FUNCTION_BLOCK FB_PrintPositionDmax EXTENDS FB_BasePrint IMPLEMENTS I_Sim
VAR_INPUT
  IlEncoderPulse      AT%I* : UDINT;                // Encoder counter intput
  IbEncoderWcState    AT%I* : BOOL;                 // Encoder EL5101 WcState
END_VAR
VAR_OUTPUT
  bStarted                  : BOOL;                 // position started moving
  bMoving                   : BOOL;                 // position is moving
END_VAR
// ----------------------------------
// configuration
VAR
  // configuration (init)
  _fPrintResolution         : LREAL := 600;         // print(head) resolution in [dpi]
  _fSubPxResolution         : LREAL := 32;          // SubPixel resolution [SubPx], resolution factor (fI_PrintResolution*fI_SubPxResolution=>Output resolution)
  _fTaskCycleTime           : LREAL := 0.002;        // Task cycle time in [s]
END_VAR
VAR PERSISTENT
  // config values changable during runtime (recipe, visu, property)
  _fEncoderResolution       : LREAL := 2.00475;     // Encoder resolution
  _bEnSpeedComp             : BOOL := FALSE;
  _fSpeedCompFactor         : LREAL := 0.0;         // TODO: define value
  _fSpeedCompRefSpeed       : LREAL := 0.0;         // TODO: define value
END_VAR
VAR CONSTANT
  fC_MinSpeed               : LREAL := 0.05;
END_VAR
// ---------------------------------
// internal variables
VAR
  // fb inst
  fbPositionMaster          : FB_PositionMaster;

  // internal vars
  fEncoderReso              : LREAL;                // used encoder resolution
  rTrigMoving               : R_TRIG;
  // simulation
  _bSim                     : BOOL;
    
  // test functions
  (*bEnTestVsOld              : BOOL;    
  fbVencoder                : FB_V_ENCODER;
  Fb_Ph_Master              : FB_POSITION_MASTER;
  *)
END_VAR

// set internal used resolution
fEncoderReso := _fEncoderResolution;  

// compensate resolution (if enabled)
IF _bEnSpeedComp THEN
  fEncoderReso := F_EncoderSpeedComp(   
    fMasterSpeed:=fbPositionMaster.fMasterSpeed,
    fResolution:=fEncoderReso,
    fSpeedCompFactor:=_fSpeedCompFactor,
    fSpeedCompRefSpeed:=_fSpeedCompRefSpeed
  );
END_IF

// calc position / speed
fbPositionMaster(fResolutionInput:=fEncoderReso, lPosReference:=IlEncoderPulse);
// postion status
bMoving := ABS(fbPositionMaster.fMasterSpeed) >= fC_MinSpeed; 
rTrigMoving(CLK:=bMoving);   // create started trigger output
bStarted := rTrigMoving.Q OR fbPositionMaster.bSyncReq;

{attribute 'monitoring' := 'call'}
(*Simulation is enabled set/get*)
PROPERTY bSimEnable : BOOL
GET
bSimEnable := _bSim;
END_GET
SET
_bSim := bSimEnable;
fbPositionMaster.bSim := _bSim;
END_SET
END_PROPERTY

(*
  Get current "default" position.
  [SubPx] as return value and [um] as output
  :return: position in SubPx resolution
*)
METHOD getPosition : DINT
VAR_OUTPUT
  nPosition_px       : DINT;                 // Master position in [px]
  fPosition_um       : LREAL;                // Master position in [um]
END_VAR
getPosition := fbPositionMaster.lMasterPosition;
nPosition_px := fbPositionMaster.lMasterPosition / LREAL_TO_DINT(_fSubPxResolution);
fPosition_um := fbPositionMaster.fMasterPosition;
END_METHOD

(*
  Get "default" speed.
*)
METHOD getSpeed : LREAL
getSpeed := fbPositionMaster.fMasterSpeed;
END_METHOD

METHOD Init : BOOL
VAR_INPUT
  fPrintResolution    : LREAL := 600;         // print(head) resolution in [dpi]
  fSubPxResolution    : LREAL := 32;          // SubPixel resolution [SubPx], resolution factor (fI_PrintResolution*fI_SubPxResolution=>Output resolution)
  fTaskCycleTime      : LREAL;                 // Task cycle time in [s]
END_VAR
// store config
_fPrintResolution := fPrintResolution;
_fSubPxResolution := fSubPxResolution;
_fTaskCycleTime   := fTaskCycleTime;

// init fbs
// - position master
fbPositionMaster.init(
  fI_PrintResolution:=fPrintResolution, 
  fI_SubPxResolution:=fSubPxResolution, 
  fI_TaskCycleTime:=fTaskCycleTime, 
  bI_HWEncoder:=FALSE
);
END_METHOD

METHOD reset
VAR_INPUT
END_VAR
// reset positioning system
fbPositionMaster.reset();
END_METHOD

END_FUNCTION_BLOCK

(* stored: Version 1.1.0.1, ProductVersion 3.1.4024.11
   POU FB_PrintPositionDmax: Id {726347b1-24f3-41dd-8d38-18de7bf18c3b}, SpecialFunc None
   Folder I_Sim: Id {bd8ec4af-70d9-4e9b-8cdc-91b3cc2e54db}
   Property bSimEnable: Id {30fe551a-b50f-4bf8-9016-a91da26e946e}
   Get Get: Id {ba61aeca-91e8-4a46-b50a-3f72adba58be}
   Set Set: Id {bfec738f-7656-45d1-b0ac-a7a5be9bcbcf}
   Method getPosition: Id {f3e3b96b-183e-4641-b112-e525c3bb6c11}
   Method getSpeed: Id {89c2b88d-36bc-48c9-87d7-952cfd236342}
   Method Init: Id {0edf7ce9-df28-43fb-8910-213c45b50fdb}
   Method reset: Id {2192cbfc-67ef-40f5-ae03-86c2f311383b} *)
